(* PLC project Counter (OSIE), Unknown Unnamed 1 *)
(* stored: creationDateTime 2021-05-14T14:33:11, modificationDateTime 2021-11-01T11:37:11 *)

FUNCTION_BLOCK CounterST
  VAR_INPUT
    Reset : BOOL;
  END_VAR
  VAR_OUTPUT
    Out1 : INT;
    Out0 : INT;
  END_VAR
  VAR
    Cnt1 : INT;
    Cnt0 : INT;
  END_VAR
  VAR_EXTERNAL
    ResetCounterValue : INT;
    Relay0 : DINT;
    Relay1 : DINT;
    Relay2 : DINT;
    Relay3 : DINT;
    Relay4 : DINT;
    Relay5 : DINT;
    Relay6 : DINT;
    Relay7 : DINT;
  END_VAR

            IF Reset THEN
  Cnt0 := ResetCounterValue;
  Cnt1 := ResetCounterValue;
  Reset := False;
ELSE
  Cnt0 := Cnt0 + 1;
  Cnt1 := Cnt1 + 1;
  IF Cnt1 = 50 THEN
    Relay0 := 1;
    Relay1 := 1; 
    Relay2 := 1;
    Relay3 := 1;
    Relay4 := 1;
    Relay5 := 1;
    Relay6 := 1;
    Relay7 := 1;
  END_IF;
  
  IF Cnt1 = 100 THEN
    Relay0 := 0;
    Relay1 := 0;
    Relay2 := 0;
    Relay3 := 0;
    Relay4 := 0;
    Relay5 := 0;
    Relay6 := 0;
    Relay7 := 0;
    Cnt1 := 0;
  END_IF;
  
END_IF;

Out1 := Cnt1;
Out0 := Cnt0;
          
END_FUNCTION_BLOCK

PROGRAM plc_prg
  VAR_INPUT
    Reset : BOOL;
  END_VAR
  VAR_OUTPUT
    Cnt0 : INT;
    Cnt1 : INT;
  END_VAR
  VAR
    CounterST0 : CounterST;
  END_VAR

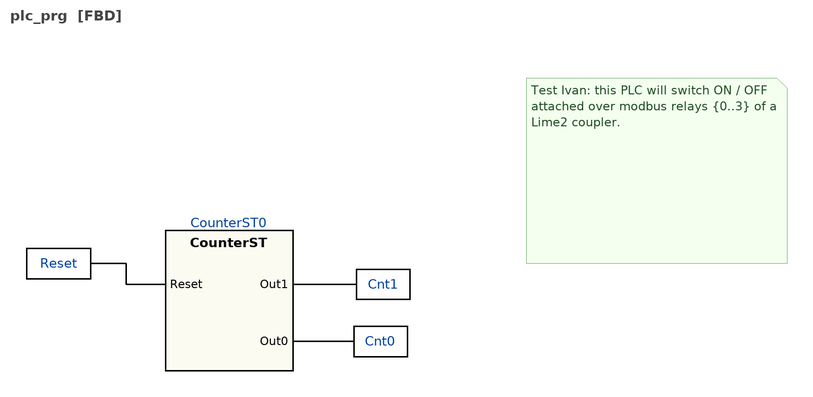
(* FBD diagram, written out as Structured Text *)
(* Test Ivan: this PLC will switch ON / OFF attached over modbus relays {0..3} of a Lime2 coupler. *)
CounterST0(Reset := Reset);
Cnt1 := CounterST0.Out1;
Cnt0 := CounterST0.Out0;
END_PROGRAM

CONFIGURATION config
  VAR_GLOBAL
    ResetCounterValue : INT := 0;
    Relay0 AT %QD1.0 : DINT := 0;  (* [I2C0] OPC-UA relay 0 *)
    Relay1 AT %QD1.1 : DINT := 0;  (* [I2C0] OPC-UA relay 1 *)
    Relay2 AT %QD1.2 : DINT := 0;  (* [I2C0] OPC-UA relay 2 *)
    Relay3 AT %QD1.3 : DINT := 0;  (* [I2C0] OPC-UA relay 2 *)
    Relay4 AT %QD1.4 : DINT := 0;  (* [I2C1] OPC-UA relay 0 *)
    Relay5 AT %QD1.5 : DINT := 0;  (* [I2C1] OPC-UA relay 1 *)
    Relay6 AT %QD1.6 : DINT := 0;  (* [I2C1] OPC-UA relay 2 *)
    Relay7 AT %QD1.7 : DINT := 0;  (* [I2C1] OPC-UA relay 3 *)
  END_VAR
  RESOURCE resource1 ON PLC
    TASK task0(INTERVAL := T#20ms, PRIORITY := 0);
    PROGRAM instance0 WITH task0 : plc_prg;
  END_RESOURCE
END_CONFIGURATION
